(* IEC 61131-3 sources: CodesysTest/export/Interfaces/IExhaustable.itf, 1 file *)

(* ---- Exhaust.m.st ---- *)
(*#-#-#-#-#-#-#-#-#-#---Declaration---#-#-#-#-#-#-#-#-#-#-#-#-#*)

METHOD Exhaust : BOOL
VAR_INPUT
END_VAR
